{attribute 'GeneratedUsingTerminal: EL2912-0000-0016'}
{attribute addProperty BoxType "EL2912-0000-0016"}
{attribute addProperty Id "Module_1_Standard_OutputAT %Q*BOOL1Module_2_Standard_OutputAT %Q*BOOL1"}
{attribute addProperty CRC "2333906029"}
{attribute addProperty Size "2"}
TYPE Outputs_8B1C946D :
STRUCT
	{attribute addProperty Name "Module_1_Standard_Output"}
	Module_1_Standard_Output AT %Q* : BOOL;
	{attribute addProperty Name "Module_2_Standard_Output"}
	Module_2_Standard_Output AT %Q* : BOOL;
END_STRUCT
END_TYPE

(* stored: Version 1.2.0.0, ProductVersion 3.1.4024.9
   DUT Outputs_8B1C946D: Id {f7a36f6a-7233-44e5-85a0-f372e8177c30} *)
